// TIA Portal V18 export
VAR_GLOBAL   // PLC tag table "AlarmsWarnings"
   "Circuit Breaker Tripped =S1-AA1-BB2" AT %I0.0 : Bool;
   "!!choice:IsSorterDoor$$" AT %M2.0 : Bool;
   "!!choice:DoorResetNecessary$$" AT %M2.1 : Bool;
END_VAR
